Staubli VAL3: onEnterEvent.pgx

program onEnterEvent(tool& x_tTool[])
begin
  //
  // NB sEvent is the selected
  // element in the LIST
  //
  call editTool(x_tTool.trsf)
  call tcp:setTool(x_tTool,nIndexTool)
  logMsg("[VALlaser] INTERFACE:Change value of the tool :"+toString("",nIndexTool))
  //
end
